(* IEC 61131-3 sources: pandora/pandora/aws-platform-main/aws-platform-main/test/Motion, 3 files *)

(* ---- AnalogAxis.st ---- *)
USING Esab.Motion.MeasurementSystem;
USING Esab.Utils.Alarming.Mock;
USING Esab.Motion.MeasurementSystems.Mock;
USING Esab.Io.Mock;
USING Esab.Utils.Timer.Mock;
USING Esab.Utils.Assets;

USING AxUnit;

NAMESPACE Esab.Motion.Test

    {TestFixture}
    CLASS AnalogAxisTests
        VAR PRIVATE
            _linearAnalogAxis : AnalogAxis;
            _rotaryAnalogAxis : AnalogAxis;
            _simulatedLinearAnalogAxis : SimulatedAnalogAxis;
            _simulatedRotaryAnalogAxis : SimulatedAnalogAxis;

            _io : AnalogAxisIo;
            _defaultIo : AnalogAxisIo;
            _runtimeParameters : AnalogAxisRuntimeParameters;
            _defaultRuntimeParameters : AnalogAxisRuntimeParameters;
            _hardwareConfiguration : AnalogAxisHardwareConfiguration;
            _defaultHardwareConfiguration : AnalogAxisHardwareConfiguration;

            _speedMeasurementTimer : OnDelayMock;
            _speedWheel : SpeedWheelMock;
            _speedAlarm : AlarmMock;

            _axis : IAxis;
            _axisAsset : REF_TO Asset;
            _observable : REF_TO AxisObservable;
        END_VAR

        {FixtureSetup}
        METHOD PUBLIC TestFixtureSetup
            _defaultRuntimeParameters.MeasuringSpeed := 10.0;
            _defaultRuntimeParameters.SpeedSettlingTime := LTIME#10s;
            _defaultRuntimeParameters.Axis.JogSpeed := 20.0;
            _defaultRuntimeParameters.Axis.JogHighSpeed := 40.0;
            _defaultRuntimeParameters.Axis.ObjectRadius := 314.15;

            _defaultHardwareConfiguration.Axis.AxisType := AxisType#Linear;
            _defaultHardwareConfiguration.MaximumSpeed := 100.0;

            _linearAnalogAxis.Setup(
                REF(_io),
                REF(_runtimeParameters),
                REF(_hardwareConfiguration),
                _speedWheel,
                _speedMeasurementTimer,
                _speedAlarm,
                NULL
            );

            _rotaryAnalogAxis.Setup(
                REF(_io),
                REF(_runtimeParameters),
                REF(_hardwareConfiguration),
                _speedWheel,
                _speedMeasurementTimer,
                _speedAlarm,
                NULL
            );

            _simulatedLinearAnalogAxis.Setup(
                REF(_runtimeParameters),
                REF(_hardwareConfiguration),
                NULL
            );

            _simulatedRotaryAnalogAxis.Setup(
                REF(_runtimeParameters),
                REF(_hardwareConfiguration),
                NULL
            );
        END_METHOD

        {TestSetup}
        METHOD PUBLIC TestSetup
            _io := _defaultIo;
            _runtimeParameters := _defaultRuntimeParameters;
            _hardwareConfiguration := _defaultHardwareConfiguration;

            _speedWheel.MockReset();
            _speedMeasurementTimer.MockReset();
            _speedAlarm.MockReset();
        END_METHOD

        {Test(axisNo := 1)}
        {Test(axisNo := 2)}
        {Test(axisNo := 3)}
        {Test(axisNo := 4)}
        METHOD PUBLIC PowerOnOff
            VAR_INPUT
                axisNo : INT;
            END_VAR

            VAR_TEMP
                _enabled : BOOL := FALSE;
            END_VAR

            THIS.SetAxis(axisNo);

            _axis.PowerOn();
            _axisAsset^.Execute();

            Assert.Equal(_axis.IsEnabled(), TRUE);
            Assert.Equal(_observable^.Enabled, TRUE);

            IF axisNo = 1 OR axisNo = 2 THEN
                _io.Outputs.RemoteControl.Write(_enabled);
                Assert.Equal(_enabled, TRUE);
            ELSE
                Assert.Equal(_axis.IsEnabled(), TRUE);
            END_IF;

            _axis.PowerOff();
            _axisAsset^.Execute();

            Assert.Equal(_observable^.Enabled, FALSE);

            IF axisNo = 1 OR axisNo = 2 THEN
                _io.Outputs.RemoteControl.Write(_enabled);
                Assert.Equal(_enabled, FALSE);
            ELSE
                Assert.Equal(_axis.IsEnabled(), FALSE);
            END_IF;
        END_METHOD

        {Test(axisNo := 1)}
        {Test(axisNo := 2)}
        {Test(axisNo := 3)}
        {Test(axisNo := 4)}
        METHOD PUBLIC AbsolutePositioning
            VAR_INPUT
                axisNo : INT;
            END_VAR

            VAR_TEMP
                _command : AxisPositioningCommand;
                _commandError : AxisCommandError;
                _speedReference : REAL;
            END_VAR

            THIS.SetAxis(axisNo);

            _axis.PowerOn();

            _command.Id := 42;
            _command.Acceleration := -1.0;
            _command.Deceleration := -1.0;
            _command.Jerk := -1.0;
            _command.PositioningDirection := AxisPositioningDirection#Positive;
            _command.CommandType := AxisCommandType#Absolute;
            _command.Position := 100.0;
            _command.Velocity := 10.0;

            _commandError := _axis.ExecutePositioningCommand(_command);

            Assert.Equal(_commandError, AxisCommandError#UnsupportedCommandType);
        END_METHOD

        {Test(axisNo := 1)}
        {Test(axisNo := 2)}
        {Test(axisNo := 3)}
        {Test(axisNo := 4)}
        METHOD PUBLIC RelativePositioning
            VAR_INPUT
                axisNo : INT;
            END_VAR

            VAR_TEMP
                _command : AxisPositioningCommand;
                _commandError : AxisCommandError;
                _speedReference : REAL;
            END_VAR

            THIS.SetAxis(axisNo);

            _axis.PowerOn();

            _command.Id := 42;
            _command.Acceleration := -1.0;
            _command.Deceleration := -1.0;
            _command.Jerk := -1.0;
            _command.PositioningDirection := AxisPositioningDirection#Positive;
            _command.CommandType := AxisCommandType#Relative;
            _command.Position := 100.0;
            _command.Velocity := 10.0;

            _commandError := _axis.ExecutePositioningCommand(_command);

            Assert.Equal(_commandError, AxisCommandError#UnsupportedCommandType);
        END_METHOD

        {Test(axisNo := 1)}
        {Test(axisNo := 2)}
        {Test(axisNo := 3)}
        {Test(axisNo := 4)}
        METHOD PUBLIC ForwardVelocity
            VAR_INPUT
                axisNo : INT;
            END_VAR

            VAR_TEMP
                _command : AxisPositioningCommand;
                _forward : BOOL;
                _reverse : BOOL;
                _speedReference : INT;
            END_VAR

            THIS.SetAxis(axisNo);

            _runtimeParameters.Axis.ObjectRadius := 750.0;

            _command.CommandType := AxisCommandType#Velocity;
            _command.Velocity := 100.0;

            _axis.PowerOn();

            Assert.Equal(_observable^.Busy, FALSE);

            _axis.ExecutePositioningCommand(_command);
            _speedWheel.GetMeasuredVelocityMock.Value := 100.0;
            _axisAsset^.Execute();

            IF axisNo = 1 OR axisNo = 2 THEN
                _io.Outputs.Forward.Write(_forward);
                _io.Outputs.Reverse.Write(_reverse);
                _io.Outputs.SpeedReference.Write(_speedReference);

                Assert.Equal(_forward, TRUE);
                Assert.Equal(_reverse, FALSE);
                Assert.Equal(_speedReference, 27648);
            END_IF;

            IF _hardwareConfiguration.Axis.AxisType = AxisType#Linear THEN
                Assert.Equal(_axis.ActualLinearVelocity(), 100.0);
                Assert.Equal(_observable^.LinearVelocity, 100.0);

                Assert.Equal(_axis.ActualAngularVelocity(), 0.0);
                Assert.Equal(_observable^.AngularVelocity, 0.0);
            ELSE
                Assert.Equal(_axis.ActualLinearVelocity(), 100.0);
                Assert.Equal(_observable^.LinearVelocity, 100.0);

                Assert.InRange(_axis.ActualAngularVelocity(), 7.63, 0.01);
                Assert.InRange(_observable^.AngularVelocity, 7.63, 0.01);
            END_IF;

            Assert.Equal(_observable^.Busy, TRUE);
        END_METHOD

        {Test(axisNo := 1)}
        {Test(axisNo := 2)}
        {Test(axisNo := 3)}
        {Test(axisNo := 4)}
        METHOD PUBLIC ReverseVelocity
            VAR_INPUT
                axisNo : INT;
            END_VAR

            VAR_TEMP
                _command : AxisPositioningCommand;
                _forward : BOOL;
                _reverse : BOOL;
                _speedReference : INT;
            END_VAR

            THIS.SetAxis(axisNo);

            _runtimeParameters.Axis.ObjectRadius := 750.0;

            _command.CommandType := AxisCommandType#Velocity;
            _command.Velocity := -100.0;

            _axis.PowerOn();

            Assert.Equal(_observable^.Busy, FALSE);

            _axis.ExecutePositioningCommand(_command);
            _speedWheel.GetMeasuredVelocityMock.Value := -100.0;
            _axisAsset^.Execute();

            IF axisNo = 1 OR axisNo = 2 THEN
                _io.Outputs.Forward.Write(_forward);
                _io.Outputs.Reverse.Write(_reverse);
                _io.Outputs.SpeedReference.Write(_speedReference);

                Assert.Equal(_forward, FALSE);
                Assert.Equal(_reverse, TRUE);
                Assert.Equal(_speedReference, 27648);
            END_IF;

            IF _hardwareConfiguration.Axis.AxisType = AxisType#Linear THEN
                Assert.Equal(_axis.ActualLinearVelocity(), -100.0);
                Assert.Equal(_observable^.LinearVelocity, -100.0);

                Assert.Equal(_axis.ActualAngularVelocity(), 0.0);
                Assert.Equal(_observable^.AngularVelocity, 0.0);
            ELSE
                Assert.Equal(_axis.ActualLinearVelocity(), -100.0);
                Assert.Equal(_observable^.LinearVelocity, -100.0);

                Assert.InRange(_axis.ActualAngularVelocity(), -7.63, 0.01);
                Assert.InRange(_observable^.AngularVelocity, -7.63, 0.01);
            END_IF;

            Assert.Equal(_observable^.Busy, TRUE);
        END_METHOD

        // Not run for simulated axis, because we currently do not mock the time accumulator.
        // So there is no way to fake the time progressing.
        {Test(axisNo := 1)}
        {Test(axisNo := 2)}
        METHOD PUBLIC Position
            VAR_INPUT
                axisNo : INT;
            END_VAR

            VAR_TEMP
                _forward : BOOL;
                _reverse : BOOL;
                _speed : INT;
            END_VAR

            THIS.SetAxis(axisNo);

            _speedWheel.GetMeasuredPositionMock.Value := 500.0;
            _runtimeParameters.Axis.ObjectRadius := 750.0;

            _axisAsset^.Execute();

            IF _hardwareConfiguration.Axis.AxisType = AxisType#Linear THEN
                Assert.Equal(_axis.ActualLinearPosition(), 500.0);
                Assert.Equal(_observable^.LinearPosition, 500.0);

                Assert.Equal(_axis.ActualAngularPosition(), 0.0);
                Assert.Equal(_observable^.AngularPosition, 0.0);
            ELSE
                Assert.Equal(_axis.ActualLinearPosition(), 500.0);
                Assert.Equal(_observable^.LinearPosition, 500.0);

                Assert.InRange(_axis.ActualAngularPosition(), 38.20, 0.01);
                Assert.InRange(_observable^.AngularPosition, 38.20, 0.01);
            END_IF;
        END_METHOD

        {Test(axisNo := 1)}
        {Test(axisNo := 2)}
        {Test(axisNo := 3)}
        {Test(axisNo := 4)}
        METHOD PUBLIC JogPositive
            VAR_INPUT
                axisNo : INT;
            END_VAR

            VAR_TEMP
                _forward : BOOL;
                _reverse : BOOL;
                _speed : INT;
            END_VAR

            THIS.SetAxis(axisNo);

            _runtimeParameters.Axis.JogSpeed := 50.0;
            _runtimeParameters.Axis.JogHighSpeed := 100.0;

            _axis.PowerOn();

            _axis.JogPositive();
            _speedWheel.GetMeasuredVelocityMock.Value := 50.0;
            _axisAsset^.Execute();

            _io.Outputs.Forward.Write(_forward);
            _io.Outputs.Reverse.Write(_reverse);
            _io.Outputs.SpeedReference.Write(_speed);

            IF axisNo = 1 OR axisNo = 2 THEN
                Assert.Equal(_forward, TRUE);
                Assert.Equal(_reverse, FALSE);
                Assert.Equal(_speed, 27648/2);
            END_IF;

            Assert.Equal(_axis.ActualLinearVelocity(), 50.0);
            Assert.Equal(_observable^.LinearVelocity, 50.0);

            _axis.JogPositive();
            _axisAsset^.Execute();
            _axis.JogPositive();
            _axisAsset^.Execute();
            _axis.JogPositive();
            _axisAsset^.Execute();
            _axis.JogPositive();
            _axisAsset^.Execute();

            _io.Outputs.Forward.Write(_forward);
            _io.Outputs.Reverse.Write(_reverse);
            _io.Outputs.SpeedReference.Write(_speed);

            IF axisNo = 1 OR axisNo = 2 THEN
                Assert.Equal(_forward, TRUE);
                Assert.Equal(_reverse, FALSE);
                Assert.Equal(_speed, 27648/2);
            END_IF;

            Assert.Equal(_axis.ActualLinearVelocity(), 50.0);
            Assert.Equal(_observable^.LinearVelocity, 50.0);

            _speedWheel.GetMeasuredVelocityMock.Value := 0.0;

            _axisAsset^.Execute(); // Execute cycle without JogPositive, check that it stops.

            _io.Outputs.Forward.Write(_forward);
            _io.Outputs.Reverse.Write(_reverse);
            _io.Outputs.SpeedReference.Write(_speed);

            IF axisNo = 1 OR axisNo = 2 THEN
                Assert.Equal(_forward, FALSE);
                Assert.Equal(_reverse, FALSE);
                Assert.Equal(_speed, 0);
            END_IF;

            Assert.Equal(_axis.ActualLinearVelocity(), 0.0);
            Assert.Equal(_observable^.LinearVelocity, 0.0);
        END_METHOD

        {Test(axisNo := 1)}
        {Test(axisNo := 2)}
        {Test(axisNo := 3)}
        {Test(axisNo := 4)}
        METHOD PUBLIC JogNegative
            VAR_INPUT
                axisNo : INT;
            END_VAR

            VAR_TEMP
                _forward : BOOL;
                _reverse : BOOL;
                _speed : INT;
            END_VAR

            THIS.SetAxis(axisNo);

            _runtimeParameters.Axis.JogSpeed := 50.0;
            _runtimeParameters.Axis.JogHighSpeed := 100.0;

            _axis.PowerOn();

            _axis.JogNegative();
            _speedWheel.GetMeasuredVelocityMock.Value := -50.0;
            _axisAsset^.Execute();

            IF axisNo = 1 OR axisNo = 2 THEN
                _io.Outputs.Forward.Write(_forward);
                _io.Outputs.Reverse.Write(_reverse);
                _io.Outputs.SpeedReference.Write(_speed);

                Assert.Equal(_forward, FALSE);
                Assert.Equal(_reverse, TRUE);
                Assert.Equal(_speed, 27648/2);
            END_IF;

            Assert.Equal(_axis.ActualLinearVelocity(), -50.0);
            Assert.Equal(_observable^.LinearVelocity, -50.0);

            _axis.JogNegative();
            _axisAsset^.Execute();
            _axis.JogNegative();
            _axisAsset^.Execute();
            _axis.JogNegative();
            _axisAsset^.Execute();
            _axis.JogNegative();
            _axisAsset^.Execute();

            _io.Outputs.Forward.Write(_forward);
            _io.Outputs.Reverse.Write(_reverse);
            _io.Outputs.SpeedReference.Write(_speed);

            IF axisNo = 1 OR axisNo = 2 THEN
                Assert.Equal(_forward, FALSE);
                Assert.Equal(_reverse, TRUE);
                Assert.Equal(_speed, 27648/2);
            END_IF;

            Assert.Equal(_axis.ActualLinearVelocity(), -50.0);
            Assert.Equal(_observable^.LinearVelocity, -50.0);

            _speedWheel.GetMeasuredVelocityMock.Value := 0.0;

            _axisAsset^.Execute(); // Execute cycle without JogPositive, check that it stops.

            _io.Outputs.Forward.Write(_forward);
            _io.Outputs.Reverse.Write(_reverse);
            _io.Outputs.SpeedReference.Write(_speed);

            IF axisNo = 1 OR axisNo = 2 THEN
                Assert.Equal(_forward, FALSE);
                Assert.Equal(_reverse, FALSE);
                Assert.Equal(_speed, 0);
            END_IF;

            Assert.Equal(_axis.ActualLinearVelocity(), 0.0);
            Assert.Equal(_observable^.LinearVelocity, 0.0);
        END_METHOD

        {Test(axisNo := 1)}
        {Test(axisNo := 2)}
        //{Test(axisNo := 3)}
        //{Test(axisNo := 4)}
        METHOD PUBLIC SpeedMonitoringAlarm
            VAR_INPUT
                axisNo : INT;
            END_VAR

            VAR_TEMP
                _command : AxisPositioningCommand;
            END_VAR

            THIS.SetAxis(axisNo);

            _command.CommandType := AxisCommandType#Velocity;
            _command.Velocity := 100.0;

            _axis.PowerOn();

            _axis.ExecutePositioningCommand(_command);
            _speedWheel.GetMeasuredVelocityMock.Value := 50.0;
            _axisAsset^.Execute();

            Assert.Equal(_speedAlarm.ExecuteMock.GetCallCount() > UINT#0, TRUE);
            Assert.Equal(_speedAlarm.ExecuteMock.SIG, TRUE);
            _speedAlarm.IsActiveMock.Value := TRUE;
            _axisAsset^.Execute();

            //Assert.Equal(_observable^.State, RollerBedState#Error);
        END_METHOD

        {Test(axisNo := 1)}
        {Test(axisNo := 2)}
        //{Test(axisNo := 3)}
        //{Test(axisNo := 4)}
        METHOD PUBLIC Calibrate
            VAR_INPUT
                axisNo : INT;
            END_VAR

            VAR_TEMP
                _measurementListener : IMeasurementSystemListener;
            END_VAR

            THIS.SetAxis(axisNo);

            _measurementListener ?= _axis;
            Assert.Equal(_measurementListener <> NULL, TRUE);

            _runtimeParameters.Axis.ObjectRadius := 1500.0;

            _speedWheel.GetMeasuredPositionMock.Value := 0.0;
            _measurementListener.ArrivedAtReferencePoint();
            _axisAsset^.Execute();

            Assert.Greater(_speedWheel.GetMeasuredPositionMock.GetCallCount(), UINT#0);

            _speedWheel.GetMeasuredPositionMock.Value := 4398.22;
            _measurementListener.ArrivedAtReferencePoint();
            _axisAsset^.Execute();

            Assert.Greater(_speedWheel.GetMeasuredPositionMock.GetCallCount(), UINT#1);
            Assert.InRange(_runtimeParameters.Axis.ObjectRadius, 700.0, 0.01);
            Assert.Equal(_axis.IsHomed(), TRUE);
            Assert.Equal(_observable^.Homed, TRUE);
        END_METHOD

        {Test(axisNo := 1)}
        {Test(axisNo := 2)}
        METHOD PUBLIC SpeedAdaptationIncreaseMax
            VAR_INPUT
                axisNo : INT;
            END_VAR

            VAR_TEMP
                _speed : INT;
                _command : AxisHomingCommand;
            END_VAR

            THIS.SetAxis(axisNo);

            _runtimeParameters.MeasuringSpeed := 5.0;
            _hardwareConfiguration.MaximumSpeed := 10.0;
            _command.HomingType := AxisHomingType#Active;

            _axis.ExecuteHomingCommand(_command);
            _speedWheel.GetMeasuredVelocityMock.Value := 10.0;
            _io.Outputs.SpeedReference.Write(_speed);
            _speedMeasurementTimer.ExpiredMock.Value := TRUE;
            Assert.Equal(_speed, 27648/2);
            _axisAsset^.Execute();
            _axisAsset^.Execute();
            _axisAsset^.Execute();
            _axisAsset^.Execute();

            Assert.Equal(_hardwareConfiguration.MaximumSpeed, 20.0);
            _io.Outputs.SpeedReference.Write(_speed);
            Assert.Equal(_speed, 27648/4);
        END_METHOD

        {Test(axisNo := 1)}
        {Test(axisNo := 2)}
        METHOD PUBLIC SpeedAdaptationDecreaseMax
            VAR_INPUT
                axisNo : INT;
            END_VAR

            VAR_TEMP
                _speed : INT;
                _command : AxisHomingCommand;
            END_VAR

            THIS.SetAxis(axisNo);

            _runtimeParameters.MeasuringSpeed := 5.0;
            _hardwareConfiguration.MaximumSpeed := 10.0;
            _command.HomingType := AxisHomingType#Active;

            _axis.ExecuteHomingCommand(_command);
            _speedWheel.GetMeasuredVelocityMock.Value := 2.5;
            _io.Outputs.SpeedReference.Write(_speed);
            _speedMeasurementTimer.ExpiredMock.Value := TRUE;
            Assert.Equal(_speed, 27648/2);
            _axisAsset^.Execute();
            _axisAsset^.Execute();
            _axisAsset^.Execute();
            _axisAsset^.Execute();

            Assert.Equal(_hardwareConfiguration.MaximumSpeed, 5.0);
            _io.Outputs.SpeedReference.Write(_speed);
            Assert.Equal(_speed, 27648);
        END_METHOD

        {Test(axisNo := 1)}
        {Test(axisNo := 2)}
        {Test(axisNo := 3)}
        {Test(axisNo := 4)}
        METHOD PUBLIC SetJogSpeed
            VAR_INPUT
                axisNo : INT;
            END_VAR

            VAR_TEMP
                _speed : INT;
                _command : AxisHomingCommand;
            END_VAR

            THIS.SetAxis(axisNo);

            _axis.SetJogSpeed(5.0);

            Assert.Equal(_runtimeParameters.Axis.JogSpeed, 5.0);
        END_METHOD

        {Test(axisNo := 1)}
        {Test(axisNo := 2)}
        {Test(axisNo := 3)}
        {Test(axisNo := 4)}
        METHOD PUBLIC SetJogHighSpeed
            VAR_INPUT
                axisNo : INT;
            END_VAR

            VAR_TEMP
                _speed : INT;
                _command : AxisHomingCommand;
            END_VAR

            THIS.SetAxis(axisNo);

            _axis.SetJogHighSpeed(10.0);

            Assert.Equal(_runtimeParameters.Axis.JogHighSpeed, 10.0);
        END_METHOD

        {Test(axisNo := 1)}
        {Test(axisNo := 2)}
        {Test(axisNo := 3)}
        {Test(axisNo := 4)}
        METHOD PUBLIC SetObjectRadius
            VAR_INPUT
                axisNo : INT;
            END_VAR

            VAR_TEMP
                _speed : INT;
                _command : AxisHomingCommand;
            END_VAR

            THIS.SetAxis(axisNo);

            _axis.SetObjectRadius(1000.0);

            Assert.Equal(_runtimeParameters.Axis.ObjectRadius, 1000.0);
        END_METHOD

        METHOD PRIVATE SetAxis
            VAR_INPUT
                axisNo : INT;
            END_VAR

            CASE axisNo OF
                1:
                    _axis := _linearAnalogAxis;
                2:
                    _hardwareConfiguration.Axis.AxisType := AxisType#Rotary;
                    _axis := _rotaryAnalogAxis;
                3:
                    _axis := _simulatedLinearAnalogAxis;
                4:
                    _hardwareConfiguration.Axis.AxisType := AxisType#Rotary;
                    _axis := _simulatedRotaryAnalogAxis;
            END_CASE;

            Assert.Equal(_axis <> NULL, TRUE);

            _axisAsset ?= _axis;
            Assert.Equal(_axisAsset <> NULL, TRUE);

            _observable ?= _axisAsset^.Observe();
            Assert.Equal(_observable <> NULL, TRUE);
        END_METHOD
    END_CLASS

END_NAMESPACE

(* ---- SpeedWheel.st ---- *)
USING Esab.Utils.Filters;
USING Esab.Io;
USING Esab.Io.Mock;
USING Esab.Motion.Mock;

USING AxUnit;
USING System.FastMath;

NAMESPACE Esab.Motion.MeasurementSystem.Test

    {TestFixture}
    CLASS SpeedWheelTests
        VAR PRIVATE
            _speedWheel : SpeedWheel;
            _hsc : HighSpeedCounterMock;
            _referenceSensor : DigitalInput;
            _hardwareConfiguration : SpeedWheelHardwareConfiguration;
            _io : SpeedWheelIo;
            _circumference : LREAL;
            _speedFilter : NoFilter;
        END_VAR

        {FixtureSetup}
        METHOD PUBLIC TestFixtureSetup
            _hardwareConfiguration.WheelDiameterInMm := LREAL#150.0;
            _hardwareConfiguration.PointsPerRevolution := UDINT#100;
            _io.ReferenceSensor := _referenceSensor;
            _speedWheel.Setup(REF(_io), REF(_hardwareConfiguration), _hsc, _speedFilter);
        END_METHOD

        {TestSetup}
        METHOD PUBLIC TestSetup
            _io.ReferenceSensor.Read(FALSE);
            _io.ReferenceSensor.Read(FALSE);

            _hsc.MockReset();
            _speedWheel.ResetMeasuredPosition();
            _circumference := Constants#PI * _hardwareConfiguration.WheelDiameterInMm;
        END_METHOD

        {Test}
        METHOD PUBLIC PositionCalculationPositiveDirection
            // One rotation of the wheel should give a full circumference worth of length units (mm).
            _hsc.GetMeasuredValueMock.Value := DINT#10;
            _hsc.GetCountValueMock.Value := DINT#0;
            _speedWheel.Execute();
            _hsc.GetCountValueMock.Value := TO_DINT(_hardwareConfiguration.PointsPerRevolution);
            _speedWheel.Execute();

            Assert.InRange(_speedWheel.GetMeasuredPosition(), _circumference, LREAL#0.0001);
        END_METHOD

        {Test}
        METHOD PUBLIC PositionCalculationNegativeDirection
            // One rotation of the wheel should give a full circumference worth of length units (mm).
            _hsc.GetMeasuredValueMock.Value := DINT#-10;
            _hsc.GetCountValueMock.Value := DINT#0;
            _speedWheel.Execute();
            _hsc.GetCountValueMock.Value := -TO_DINT(_hardwareConfiguration.PointsPerRevolution);
            _speedWheel.Execute();

            Assert.InRange(_speedWheel.GetMeasuredPosition(), -_circumference, LREAL#0.0001);
        END_METHOD

        {Test}
        METHOD PUBLIC CounterRolloverPositive
            _hsc.GetUpperCountingLimitMock.Value := 200;
            _hsc.GetLowerCountingLimitMock.Value := -200;

            // Rolling over should still increase the measured position
            _hsc.GetCountValueMock.Value := DINT#150;
            _speedWheel.ResetMeasuredPosition();
            _hsc.GetMeasuredValueMock.Value := DINT#10;
            _speedWheel.Execute();
            _hsc.GetCountValueMock.Value := DINT#-150;
            _speedWheel.Execute();

            Assert.InRange(_speedWheel.GetMeasuredPosition(), _circumference, LREAL#0.0001);
        END_METHOD

        {Test}
        METHOD PUBLIC CounterRolloverNegative
            _hsc.GetUpperCountingLimitMock.Value := 200;
            _hsc.GetLowerCountingLimitMock.Value := -200;

            // Rolling over should still increase the measured position
            _hsc.GetCountValueMock.Value := DINT#-150;
            _speedWheel.ResetMeasuredPosition();
            _hsc.GetMeasuredValueMock.Value := DINT#-10;
            _speedWheel.Execute();
            _hsc.GetCountValueMock.Value := DINT#150;
            _speedWheel.Execute();

            Assert.InRange(_speedWheel.GetMeasuredPosition(), -_circumference, LREAL#0.0001);
        END_METHOD

        {Test}
        METHOD PUBLIC Speed
            _hsc.GetMeasuredValueMock.Value := DINT#100;

            _speedWheel.Execute();

            Assert.Equal(_speedWheel.GetMeasuredVelocity(), 100.0 * (150.0 * Constants#PI / 100));
        END_METHOD
    END_CLASS

END_NAMESPACE

(* ---- WeldHeadManipulator.st ---- *)
USING Esab.Motion.Mock;
USING Esab.Utils.Assets;
USING Esab.Hmi.Modules;
USING Esab.Utils.Timer.Mock;
USING AxUnit;
USING System.FastMath;

NAMESPACE Esab.Motion.Test

    {TestFixture}
    CLASS WeldHeadManipulatorTests
        VAR PRIVATE
            _manipulator : WeldHeadManipulator;
            _runtimeParameters : WeldHeadManipulatorRuntimeParameters;
            _hardwareConfiguration : WeldHeadManipulatorHardwareConfiguration;

            _joystick : DiscreteJoystick;
            _joystickIo : DiscreteJoystickIo;
            _joystickTimer : OnDelayMock;

            _horizontalSlide : ToPosAxisMock;
            _verticalSlide : ToPosAxisMock;
            _assetsManager : AssetsManager;
        END_VAR

        {FixtureSetup}
        METHOD PUBLIC TestFixtureSetup
            _joystick.Setup(REF(_joystickIo), _joystickTimer);
            _joystick.SetIdentifier(AssetIdentifier#P_Joystick_MotionJoystick);
            _assetsManager.RegisterAsset(REF(_joystick));

            _horizontalSlide.SetIdentifier(Esab.AssetIdentifier#HorizontalSlideAxis);
            _assetsManager.RegisterAsset(REF(_horizontalSlide));

            _verticalSlide.SetIdentifier(Esab.AssetIdentifier#VerticalSlideAxis);
            _assetsManager.RegisterAsset(REF(_verticalSlide));

            _manipulator.Setup(REF(_runtimeParameters), REF(_hardwareConfiguration), _assetsManager);
        END_METHOD

        {TestSetup}
        METHOD PUBLIC TestSetup
            _horizontalSlide.MockReset();
            _verticalSlide.MockReset();
            _manipulator.Disable();
        END_METHOD

        {Test}
        METHOD PUBLIC EnableDisable
            _horizontalSlide.IsEnabledMock.Value := TRUE;
            _verticalSlide.IsEnabledMock.Value := TRUE;

            Assert.Equal(_assetsManager.RequestAssetHandle(NULL, Esab.AssetIdentifier#HorizontalSlideAxis) <> NULL, TRUE);
            Assert.Equal(_assetsManager.RequestAssetHandle(NULL, Esab.AssetIdentifier#VerticalSlideAxis) <> NULL, TRUE);

            Assert.Equal(_manipulator.Enable(), WeldHeadManipulatorErrorCode#NoError);

            Assert.Equal(_assetsManager.RequestAssetHandle(NULL, Esab.AssetIdentifier#HorizontalSlideAxis) = NULL, TRUE);
            Assert.Equal(_assetsManager.RequestAssetHandle(NULL, Esab.AssetIdentifier#VerticalSlideAxis) = NULL, TRUE);
            Assert.Equal(_manipulator.IsEnabled(), TRUE);

            _manipulator.Disable();

            Assert.Equal(_assetsManager.RequestAssetHandle(NULL, Esab.AssetIdentifier#HorizontalSlideAxis) <> NULL, TRUE);
            Assert.Equal(_assetsManager.RequestAssetHandle(NULL, Esab.AssetIdentifier#VerticalSlideAxis) <> NULL, TRUE);
            Assert.Equal(_manipulator.IsEnabled(), FALSE);

            Assert.Equal(_manipulator.Enable(), WeldHeadManipulatorErrorCode#NoError);

            Assert.Equal(_assetsManager.RequestAssetHandle(NULL, Esab.AssetIdentifier#HorizontalSlideAxis) = NULL, TRUE);
            Assert.Equal(_assetsManager.RequestAssetHandle(NULL, Esab.AssetIdentifier#VerticalSlideAxis) = NULL, TRUE);
            Assert.Equal(_manipulator.IsEnabled(), TRUE);

            _manipulator.Disable();

            Assert.Equal(_assetsManager.RequestAssetHandle(NULL, Esab.AssetIdentifier#HorizontalSlideAxis) <> NULL, TRUE);
            Assert.Equal(_assetsManager.RequestAssetHandle(NULL, Esab.AssetIdentifier#VerticalSlideAxis) <> NULL, TRUE);
            Assert.Equal(_manipulator.IsEnabled(), FALSE);
        END_METHOD

        {Test(speed := 10.0, x_act_pos := 0.0, x_pos := 11.0, z_act_pos := 0.0, z_pos := 7.0)}
        {Test(speed := 10.0, x_act_pos := 0.0, x_pos := 11.0, z_act_pos := 0.0, z_pos := -7.0)}
        {Test(speed := 10.0, x_act_pos := 0.0, x_pos := -11.0, z_act_pos := 0.0, z_pos := 7.0)}
        {Test(speed := 10.0, x_act_pos := 0.0, x_pos := -11.0, z_act_pos := 0.0, z_pos := -7.0)}
        {Test(speed := 10.0, x_act_pos := 20.0, x_pos := 25.0, z_act_pos := 20.0, z_pos := 25.0)}
        {Test(speed := 10.0, x_act_pos := 20.0, x_pos := 25.0, z_act_pos := 20.0, z_pos := 15.0)}
        {Test(speed := 10.0, x_act_pos := 20.0, x_pos := 15.0, z_act_pos := 20.0, z_pos := 25.0)}
        {Test(speed := 10.0, x_act_pos := 20.0, x_pos := 15.0, z_act_pos := 20.0, z_pos := 15.0)}
        METHOD PUBLIC Positioning
            VAR_INPUT
                speed : LREAL;
                x_act_pos : LREAL;
                x_pos : LREAL;
                z_act_pos : LREAL;
                z_pos : LREAL;
            END_VAR

            VAR_TEMP
                position : ARRAY [0..1] OF LREAL;
                distance : ARRAY [0..1] OF LREAL;
                x_vel : LREAL;
                z_vel : LREAL;
            END_VAR

            position[0] := x_pos;
            position[1] := z_pos;

            distance[0] := Abs(x_pos - x_act_pos);
            distance[1] := Abs(z_pos - z_act_pos);

            _horizontalSlide.ActualLinearPositionMock.Value := x_act_pos;
            _verticalSlide.ActualLinearPositionMock.Value := z_act_pos;

            _manipulator.Enable();

            Assert.Equal(_horizontalSlide.ExecutePositioningCommandMock.GetCallCount(), UINT#1);
            Assert.Equal(_verticalSlide.ExecutePositioningCommandMock.GetCallCount(), UINT#1);

            // Assert that we issued a command to move the axis to their current position.
            Assert.Equal(_horizontalSlide.ExecutePositioningCommandMock.Command.CommandType, AxisCommandType#Absolute);
            Assert.Equal(_horizontalSlide.ExecutePositioningCommandMock.Command.Position, x_act_pos);

            Assert.Equal(_verticalSlide.ExecutePositioningCommandMock.Command.CommandType, AxisCommandType#Absolute);
            Assert.Equal(_verticalSlide.ExecutePositioningCommandMock.Command.Position, z_act_pos);

            // Set new target positions
            _manipulator.Move(position, speed);

            Assert.Equal(_horizontalSlide.ExecutePositioningCommandMock.GetCallCount(), UINT#2);
            Assert.Equal(_verticalSlide.ExecutePositioningCommandMock.GetCallCount(), UINT#2);

            Assert.Equal(_horizontalSlide.ExecutePositioningCommandMock.Command.CommandType, AxisCommandType#Absolute);
            Assert.Equal(_horizontalSlide.ExecutePositioningCommandMock.Command.Position, x_pos);

            Assert.Equal(_verticalSlide.ExecutePositioningCommandMock.Command.CommandType, AxisCommandType#Absolute);
            Assert.Equal(_verticalSlide.ExecutePositioningCommandMock.Command.Position, z_pos);

            // Assert that the axis will arrive at target position at the same time
            x_vel := _horizontalSlide.ExecutePositioningCommandMock.Command.Velocity;
            z_vel := _verticalSlide.ExecutePositioningCommandMock.Command.Velocity;
            Assert.InRange(distance[0]/x_vel, distance[1]/z_vel, 0.1); // It is acceptable if they are calculated to arrive within 0.1s of each other.
        END_METHOD

        {Test(speed := 10.0, x_act_pos := 0.0, x_pos := 11.0)}
        METHOD PUBLIC PositionHorizontalOnly
            VAR_INPUT
                speed : LREAL;
                x_act_pos : LREAL;
                x_pos : LREAL;
            END_VAR

            VAR_TEMP
                position : ARRAY [0..1] OF LREAL;
                distance : ARRAY [0..1] OF LREAL;
                x_vel : LREAL;
                z_act_pos : LREAL := 10.0;
            END_VAR

            position[0] := x_pos;
            position[1] := z_act_pos;

            distance[0] := Abs(x_pos - x_act_pos);
            distance[1] := 0.0;

            _horizontalSlide.ActualLinearPositionMock.Value := x_act_pos;
            _verticalSlide.ActualLinearPositionMock.Value := z_act_pos;

            _manipulator.Enable();

            _manipulator.Move(position, speed);

            Assert.Equal(_horizontalSlide.ExecutePositioningCommandMock.GetCallCount(), UINT#2);
            Assert.Equal(_verticalSlide.ExecutePositioningCommandMock.GetCallCount(), UINT#2);

            Assert.Equal(_horizontalSlide.ExecutePositioningCommandMock.Command.CommandType, AxisCommandType#Absolute);
            Assert.Equal(_horizontalSlide.ExecutePositioningCommandMock.Command.Position, x_pos);
            Assert.Equal(_horizontalSlide.ExecutePositioningCommandMock.Command.Velocity, speed);

            Assert.Equal(_verticalSlide.ExecutePositioningCommandMock.Command.CommandType, AxisCommandType#Absolute);
            Assert.Equal(_verticalSlide.ExecutePositioningCommandMock.Command.Position, z_act_pos);
        END_METHOD

        {Test(x_pos := 11.0, z_pos := 7.0, x_speed := 10.0, z_speed := 5.0)}
        METHOD PUBLIC MoveNonInterpolated
            VAR_INPUT
                x_speed : LREAL;
                z_speed : LREAL;
                x_pos : LREAL;
                z_pos : LREAL;
            END_VAR

            VAR_TEMP
                position : ARRAY [0..1] OF LREAL;
                speed : ARRAY [0..1] OF LREAL;
            END_VAR

            position[0] := x_pos;
            position[1] := z_pos;

            speed[0] := x_speed;
            speed[1] := z_speed;

            _horizontalSlide.ActualLinearPositionMock.Value := 0.0;
            _verticalSlide.ActualLinearPositionMock.Value := 0.0;

            _manipulator.Enable();
            _manipulator.SetControlMode(WeldHeadManipulatorControlMode#MoveToPosition);

            Assert.Equal(_horizontalSlide.ExecutePositioningCommandMock.GetCallCount(), UINT#1);
            Assert.Equal(_verticalSlide.ExecutePositioningCommandMock.GetCallCount(), UINT#1);

            // Assert that we issued a command to move the axis to their current position.
            Assert.Equal(_horizontalSlide.ExecutePositioningCommandMock.Command.CommandType, AxisCommandType#Absolute);
            Assert.Equal(_horizontalSlide.ExecutePositioningCommandMock.Command.Position, 0.0);

            Assert.Equal(_verticalSlide.ExecutePositioningCommandMock.Command.CommandType, AxisCommandType#Absolute);
            Assert.Equal(_verticalSlide.ExecutePositioningCommandMock.Command.Position, 0.0);

            // Set new target positions
            _manipulator.Move(position, speed);

            Assert.Equal(_horizontalSlide.ExecutePositioningCommandMock.GetCallCount(), UINT#2);
            Assert.Equal(_verticalSlide.ExecutePositioningCommandMock.GetCallCount(), UINT#2);

            Assert.Equal(_horizontalSlide.ExecutePositioningCommandMock.Command.CommandType, AxisCommandType#Absolute);
            Assert.Equal(_horizontalSlide.ExecutePositioningCommandMock.Command.Position, x_pos);
            Assert.Equal(_horizontalSlide.ExecutePositioningCommandMock.Command.Velocity, x_speed);

            Assert.Equal(_verticalSlide.ExecutePositioningCommandMock.Command.CommandType, AxisCommandType#Absolute);
            Assert.Equal(_verticalSlide.ExecutePositioningCommandMock.Command.Position, z_pos);
            Assert.Equal(_verticalSlide.ExecutePositioningCommandMock.Command.Velocity, z_speed);
        END_METHOD

        METHOD PRIVATE Execute
            _assetsManager.Execute();
            _manipulator.Execute();
        END_METHOD

        {Test(position := 1)}
        {Test(position := 2)}
        {Test(position := 3)}
        {Test(position := 4)}
        METHOD PUBLIC JoystickJogOfWeldHeadManipulator
            VAR_INPUT
                position : INT;
            END_VAR

            VAR_TEMP
                asset : REF_TO Asset;
                joystickPosition : JoystickPosition;
            END_VAR

            _manipulator.Execute();
            _manipulator.SetControlMode(WeldHeadManipulatorControlMode#JoystickJog);
            _manipulator.Enable();

            joystickPosition := position;

            // Trigger long hold callback
            CASE joystickPosition OF
                JoystickPosition#Up:
                    _joystickIo.Up.Read(TRUE);
                JoystickPosition#Down:
                    _joystickIo.Down.Read(TRUE);
                JoystickPosition#Triangle:
                    _joystickIo.Triangle.Read(TRUE);
                JoystickPosition#Square:
                    _joystickIo.Square.Read(TRUE);
            END_CASE;

            THIS.Execute();
            CASE joystickPosition OF
                JoystickPosition#Up:
                    Assert.Equal(_verticalSlide.JogPositiveMock.GetCallCount(), UINT#1);
                JoystickPosition#Down:
                    Assert.Equal(_verticalSlide.JogNegativeMock.GetCallCount(), UINT#1);
                JoystickPosition#Triangle:
                    Assert.Equal(_horizontalSlide.JogNegativeMock.GetCallCount(), UINT#1);
                JoystickPosition#Square:
                    Assert.Equal(_horizontalSlide.JogPositiveMock.GetCallCount(), UINT#1);
            END_CASE;

            THIS.Execute();
            THIS.Execute();
            THIS.Execute();
            THIS.Execute();

            CASE joystickPosition OF
                JoystickPosition#Up:
                    Assert.Equal(_verticalSlide.JogPositiveMock.GetCallCount(), UINT#5);
                JoystickPosition#Down:
                    Assert.Equal(_verticalSlide.JogNegativeMock.GetCallCount(), UINT#5);
                JoystickPosition#Triangle:
                    Assert.Equal(_horizontalSlide.JogNegativeMock.GetCallCount(), UINT#5);
                JoystickPosition#Square:
                    Assert.Equal(_horizontalSlide.JogPositiveMock.GetCallCount(), UINT#5);
            END_CASE;

            CASE joystickPosition OF
                JoystickPosition#Up:
                    _joystickIo.Up.Read(FALSE);
                JoystickPosition#Down:
                    _joystickIo.Down.Read(FALSE);
                JoystickPosition#Triangle:
                    _joystickIo.Triangle.Read(FALSE);
                JoystickPosition#Square:
                    _joystickIo.Square.Read(FALSE);
            END_CASE;
            _joystickTimer.MockReset();

            THIS.Execute();

            CASE joystickPosition OF
                JoystickPosition#Up:
                    Assert.Equal(_verticalSlide.JogPositiveMock.GetCallCount(), UINT#5);
                JoystickPosition#Down:
                    Assert.Equal(_verticalSlide.JogNegativeMock.GetCallCount(), UINT#5);
                JoystickPosition#Triangle:
                    Assert.Equal(_horizontalSlide.JogNegativeMock.GetCallCount(), UINT#5);
                JoystickPosition#Square:
                    Assert.Equal(_horizontalSlide.JogPositiveMock.GetCallCount(), UINT#5);
            END_CASE;

            _manipulator.SetControlMode(WeldHeadManipulatorControlMode#MoveToPosition);
        END_METHOD

    END_CLASS
END_NAMESPACE
